// TwinCAT 3 PLC project PRG_Test_MachineControl
// ProgramVersion: 3.1.4024.0
// libraries:
//   B_Base, * (RafalOS)
//   B_IO, * (RafalOS)
//   B_MachineControl, * (RafalOS)
//   B_StatesAndModes, * (RafalOS)
//   Tc2_Standard, * (Beckhoff Automation GmbH)
//   Tc2_System, * (Beckhoff Automation GmbH)
//   Tc3_Module, * (Beckhoff Automation GmbH)
//   TcUnit, * (www.tcunit.org)
// project tree:
//   GVLs/ GVL_TestMCSafety.TcGVL, GVL_TestRequeestChange.TcGVL, GVL_TestSystemVariable.TcGVL, GVL_TopElement1.TcGVL, GVL_TopElement2.TcGVL, GVL_TestSaMContoller.TcGVL (not stored)
//   / PlcTask.TcTTO (not stored)
//   POUs/ FB_MyDefaultConfiguration.TcPOU, FB_MachineControl_NoneTE_Test.TcPOU, FB_MyNewConfigurationAddTE.TcPOU (not stored), FB_SaMControllerTest.TcPOU
//   POUs/POUs TopElement1/ FB_ControlElement1.TcPOU (not stored), FB_ControlElement2.TcPOU (not stored), FB_TopElement1.TcPOU, ITF_ControlElement1.TcIO (not stored), ITF_ControlElement2.TcIO (not stored), ITF_TopElement1.TcIO (not stored)
//   POUs/POUs TopElement2/ FB_ControlElement3.TcPOU (not stored), FB_ControlElement5.TcPOU, FB_ControlElement4.TcPOU (not stored), FB_ControlElement6.TcPOU, FB_GroupElement1.TcPOU, FB_TopElement2.TcPOU (not stored), ITF_ControlElement3.TcIO (not stored), ITF_ControlElement5.TcIO (not stored), ITF_ControlElement4.TcIO, ITF_ControlElement6.TcIO, ITF_GroupElement1.TcIO (not stored), ITF_TopElement2.TcIO (not stored)
//   TESTs/ PRG_Test.TcPOU (not stored)

// ---- GVLs/GVL_TestMCSafety.TcGVL
{attribute 'qualified_only'}
VAR_GLOBAL
	flSS1				: FB_BaseFlag;
	flSTO				: FB_BaseFlag;
	
END_VAR

// ---- GVLs/GVL_TestRequeestChange.TcGVL
{attribute 'qualified_only'}
VAR_GLOBAL
//Przyciski zmaiany stanu	
//	fbprUndefined			: FB_RequestChanges;
	fbprAbort				: FB_MCRequiredChange;
  	fbprClear				: FB_MCRequiredChange;
   	fbprReset				: FB_MCRequiredChange;
   	fbprStart				: FB_MCRequiredChange;
   	fbprStop				: FB_MCRequiredChange;
   	fbprHold				: FB_MCRequiredChange;
   	fbprUnhold				: FB_MCRequiredChange;
   	fbprSuspend				: FB_MCRequiredChange;
   	fbprUnsuspend			: FB_MCRequiredChange;
  	fbprComplete			: FB_MCRequiredChange;
//przyciski zmiany trybu
//	fbprNiedozwolony		: FB_SITP_PolecenieZmianyTrybu (ePolecenie := E_SITP_PolecenieZmianyTrybu.brak);     
	fbprProduction			: FB_MCRequiredChange;
    fbprMaintenance			: FB_MCRequiredChange;
    fbprManual				: FB_MCRequiredChange;
    fbprWashing				: FB_MCRequiredChange;
    fbprDiagnostics			: FB_MCRequiredChange;
//    fbprUzytkownika2		: FB_RequestChanges;
//   fbprUzytkownika3		: FB_RequestChanges;
//    fbprUzytkownika4		: FB_RequestChanges;
//    fbprUzytkownika5		: FB_RequestChanges;

END_VAR

// ---- GVLs/GVL_TestSystemVariable.TcGVL
{attribute 'qualified_only'}
VAR_GLOBAL
	fbTime							: FB_BaseTime;
	fbLocation						: FB_BaseLocation;
	fbLogger						: FB_BaseLogger;
	
	stCommonData					: ST_BaseCommonData;

	fbDefaultMachineConfiguration	: FB_MyDefaultConfiguration;
	fbMachineConfigure				: FB_MCMachineConfigure;
	
	fbSaMController					: FB_SaMController;
	
	fbMachineControl				: FB_MCMachineControl;
	
END_VAR

// ---- GVLs/GVL_TopElement1.TcGVL
{attribute 'qualified_only'}
VAR_GLOBAL
	senControlElement1Start		: FB_IOSensor_NO;
	senControlElement1End		: FB_IOSensor_NO;
	fbControlElement1			: FB_ControlElement1 (
									itfsenStart	:= senControlElement1Start,
	                                itfsenEnd	:= senControlElement1End
								);
	senControlElement2Start		: FB_IOSensor_NO;
	senControlElement2End		: FB_IOSensor_NO;
	senControlElement2Position1	: FB_IOSensor_NO;
	senControlElement2Position2	: FB_IOSensor_NO;
	fbControlElement2			:  FB_ControlElement2 (
									itfsenStart		:= senControlElement2Start,
	                                itfsenEnd		:= senControlElement2End,
	                                itfsenPosition1	:= senControlElement2Position1,
								    itfsenPosition2	:= senControlElement2Position2
								);

	senTopElement1Position1		: FB_IOSensor_NO;
	senTopElement1Position2		: FB_IOSensor_NO;
	fbTopElement1				: FB_TopElement1 (
									itfControlElement1		:= fbControlElement1,
								    itfControlElement2		:= fbControlElement2,
		                           	itfsenElementPosition1	:= senTopElement1Position1,
                                    itfsenElementPosition2	:= senTopElement1Position2
								);
END_VAR

// ---- GVLs/GVL_TopElement2.TcGVL
{attribute 'qualified_only'}
VAR_GLOBAL
	senControlElement3Start		: FB_IOSensor_NO;
	senControlElement3End		: FB_IOSensor_NO;
	fbControlElement3			: FB_ControlElement3 (
									itfsenStart	:= senControlElement3Start,
	                                itfsenEnd	:= senControlElement3End
								);
	senControlElement4Start		: FB_IOSensor_NO;
	senControlElement4End		: FB_IOSensor_NO;
	senControlElement4Position1	: FB_IOSensor_NO;
	senControlElement4Position2	: FB_IOSensor_NO;
	fbControlElement4			:  FB_ControlElement4 (
									itfsenStart		:= senControlElement4Start,
	                                itfsenEnd		:= senControlElement4End,
	                                itfsenPosition1	:= senControlElement4Position1,
								    itfsenPosition2	:= senControlElement4Position2
								);

	senGroupElement1Position1	: FB_IOSensor_NO;
	senGroupElement1Position2	: FB_IOSensor_NO;
	fbGroupElement1				: FB_GroupElement1 (
									itfControlElement3	:= fbControlElement3,
								    itfControlElement4	:= fbControlElement4,
								    itfsenPosition1		:= senGroupElement1Position1,
								    itfsenPosition2		:= senGroupElement1Position2
								);

	senControlElement5Start		: FB_IOSensor_NO;
	senControlElement5End		: FB_IOSensor_NO;
	fbControlElement5			: FB_ControlElement5 (
									itfsenStart	:= senControlElement5Start,
	                                itfsenEnd	:= senControlElement5End
								);
	senControlElement6Start		: FB_IOSensor_NO;
	senControlElement6End		: FB_IOSensor_NO;
	senControlElement6Position1	: FB_IOSensor_NO;
	senControlElement6Position2	: FB_IOSensor_NO;
	fbControlElement6			:  FB_ControlElement6 (
									itfsenStart		:= senControlElement6Start,
	                                itfsenEnd		:= senControlElement6End,
	                                itfsenPosition1	:= senControlElement6Position1,
								    itfsenPosition2	:= senControlElement6Position2
								);
								
								
	senTopElement1Position1		: FB_IOSensor_NO;
	senTopElement1Position2		: FB_IOSensor_NO;
	fbTopElement2				: FB_TopElement2 (
									itfGroupElement1		:= fbGroupElement1,
									itfControlElement5		:= fbControlElement5,
								    itfControlElement6		:= fbControlElement6,
		                           	itfsenElementPosition1	:= senTopElement1Position1,
                                    itfsenElementPosition2	:= senTopElement1Position2
								);
END_VAR

// ---- POUs/POUs TopElement2/ITF_ControlElement4.TcIO
INTERFACE ITF_ControlElement4 EXTENDS ITF_BaseControlElement

END_INTERFACE

// ---- POUs/POUs TopElement2/ITF_ControlElement6.TcIO
INTERFACE ITF_ControlElement6 EXTENDS ITF_BaseControlElement

END_INTERFACE

// ---- POUs/FB_MyDefaultConfiguration.TcPOU
FUNCTION_BLOCK FB_MyDefaultConfiguration EXTENDS FB_Base IMPLEMENTS ITF_MCConfiguration
VAR

END_VAR

METHOD PUBLIC AddTopElementToLogger : BOOL
VAR_INPUT
END_VAR
GVL_TestSystemVariable.fbMachineControl.JoinTheLogger ();
END_METHOD

(*			
	RafalOS
	Rafał Osajda		29.10.2025		TC 4024.66
	Dodawanie TopElementu do systemu
*)
METHOD PUBLIC AddTopElementToMachineControl : BOOL
VAR_INPUT
	itfMachineControl			: ITF_MCMachineControlConfigure;
END_VAR
THIS^.SetText (eLocation := E_BaseLocation.pl, wsDescription := "System");
THIS^.SetText (eLocation := E_BaseLocation.en, wsDescription := "System");
THIS^.SetText (eLocation := E_BaseLocation.de, wsDescription := "System");
GVL_TestSystemVariable.fbMachineControl.SetName (stName := THIS^.GetTexts ());
itfMachineControl.AddTopElementFromConfiguration (fbTopElement	:= GVL_TestSystemVariable.fbMachineControl);
END_METHOD

METHOD PUBLIC SetStartMode : BOOL
VAR_INPUT
	itfMachineControl			: ITF_MCMachineControlConfigure;
END_VAR
itfMachineControl.SetStartMode (eStartMode := E_BaseMachineMode.Production);
END_METHOD

METHOD StateAndModes : BOOL
VAR_INPUT
	itfMachineControl			: ITF_MCMachineControlConfigure;
END_VAR
itfMachineControl.AddRequestStateChange (iNumberOfRequest := E_SaMCommandChangeState.Clear,		itfRequest := GVL_TestRequeestChange.fbprClear);
itfMachineControl.AddRequestStateChange (iNumberOfRequest := E_SaMCommandChangeState.Reset, 	itfRequest := GVL_TestRequeestChange.fbprReset);
itfMachineControl.AddRequestStateChange (iNumberOfRequest := E_SaMCommandChangeState.Start, 	itfRequest := GVL_TestRequeestChange.fbprStart);
itfMachineControl.AddRequestStateChange (iNumberOfRequest := E_SaMCommandChangeState.Stop, 		itfRequest := GVL_TestRequeestChange.fbprStop);
itfMachineControl.AddRequestStateChange (iNumberOfRequest := E_SaMCommandChangeState.Suspend, 	itfRequest := GVL_TestRequeestChange.fbprSuspend);
itfMachineControl.AddRequestStateChange (iNumberOfRequest := E_SaMCommandChangeState.Unsuspend, itfRequest := GVL_TestRequeestChange.fbprUnsuspend);
itfMachineControl.AddRequestStateChange (iNumberOfRequest := E_SaMCommandChangeState.Hold, 		itfRequest := GVL_TestRequeestChange.fbprHold);
itfMachineControl.AddRequestStateChange (iNumberOfRequest := E_SaMCommandChangeState.Unhold, 	itfRequest := GVL_TestRequeestChange.fbprUnhold);
itfMachineControl.AddRequestStateChange (iNumberOfRequest := E_SaMCommandChangeState.Complete, 	itfRequest := GVL_TestRequeestChange.fbprComplete);
itfMachineControl.AddRequestStateChange (iNumberOfRequest := E_SaMCommandChangeState.Abort,		itfRequest := GVL_TestRequeestChange.fbprAbort);

itfMachineControl.AddRequestModeChange (iNumberOfRequest := E_SaMCommandChangeMode.Production, 	itfRequest := GVL_TestRequeestChange.fbprProduction);
itfMachineControl.AddRequestModeChange (iNumberOfRequest := E_SaMCommandChangeMode.Maintenance,	itfRequest := GVL_TestRequeestChange.fbprMaintenance);
itfMachineControl.AddRequestModeChange (iNumberOfRequest := E_SaMCommandChangeMode.Manual, 		itfRequest := GVL_TestRequeestChange.fbprManual);
itfMachineControl.AddRequestModeChange (iNumberOfRequest := E_SaMCommandChangeMode.Washing,		itfRequest := GVL_TestRequeestChange.fbprWashing);
itfMachineControl.AddRequestModeChange (iNumberOfRequest := E_SaMCommandChangeMode.Diagnostisc,	itfRequest := GVL_TestRequeestChange.fbprDiagnostics);
END_METHOD

END_FUNCTION_BLOCK

// ---- POUs/POUs TopElement1/FB_TopElement1.TcPOU
FUNCTION_BLOCK FB_TopElement1 EXTENDS FB_BaseTopElement IMPLEMENTS ITF_TopElement1
VAR
	itfControlElement1		: ITF_ControlElement1;
	itfControlElement2		: ITF_ControlElement2;
	itfsenElementPosition1	: ITF_IOSensor;
	itfsenElementPosition2	: ITF_IOSensor;
END_VAR

METHOD FB_init : BOOL
VAR_INPUT
	bInitRetains : BOOL; // if TRUE, the retain variables are initialized (warm start / cold start)
	bInCopyCode : BOOL;  // if TRUE, the instance afterwards gets moved into the copy code (online change)
	itfControlElement1		: ITF_ControlElement1;
	itfControlElement2		: ITF_ControlElement2;
	itfsenElementPosition1	: ITF_IOSensor;
	itfsenElementPosition2	: ITF_IOSensor;
END_VAR
THIS^.itfControlElement1			:= itfControlElement1;
THIS^.AddControlElement (itfControlElement	:= itfControlElement1);
THIS^.SetText (eLocation 			:= E_BaseLocation.pl, wsDescription := "Nazwa controlelementu 1 pl");
THIS^.SetText (eLocation 			:= E_BaseLocation.en, wsDescription := "Nazwa controlelementu 1 en");
THIS^.SetText (eLocation 			:= E_BaseLocation.de, wsDescription := "Nazwa controlelementu 1 de");
THIS^.itfControlElement1.SetName (stName	:= THIS^.GetTexts ());

THIS^.itfControlElement2			:= itfControlElement2;
THIS^.AddControlElement (itfControlElement	:= itfControlElement2);
THIS^.SetText (eLocation 			:= E_BaseLocation.pl, wsDescription := "Nazwa controlelementu 2 pl");
THIS^.SetText (eLocation 			:= E_BaseLocation.en, wsDescription := "Nazwa controlelementu 2 en");
THIS^.SetText (eLocation 			:= E_BaseLocation.de, wsDescription := "Nazwa controlelementu 2 de");
THIS^.itfControlElement2.SetName (stName	:= THIS^.GetTexts ());

THIS^.itfsenElementPosition1		:= itfsenElementPosition1;
THIS^.AddComponent (itfComponent	:= itfsenElementPosition1);
THIS^.SetText (eLocation 			:= E_BaseLocation.pl, wsDescription := "Nazwa komponentu 1 pl");
THIS^.SetText (eLocation 			:= E_BaseLocation.en, wsDescription := "Nazwa komponentu 1 en");
THIS^.SetText (eLocation 			:= E_BaseLocation.de, wsDescription := "Nazwa komponentu 1 de");
THIS^.itfsenElementPosition1.SetName (stName	:= THIS^.GetTexts ());

THIS^.itfsenElementPosition2		:= itfsenElementPosition2;
THIS^.AddComponent (itfComponent	:= itfsenElementPosition2);
THIS^.SetText (eLocation 			:= E_BaseLocation.pl, wsDescription := "Nazwa komponentu 2 pl");
THIS^.SetText (eLocation 			:= E_BaseLocation.en, wsDescription := "Nazwa komponentu 2 en");
THIS^.SetText (eLocation 			:= E_BaseLocation.de, wsDescription := "Nazwa komponentu 2 de");
THIS^.itfsenElementPosition2.SetName (stName	:= THIS^.GetTexts ());
END_METHOD

END_FUNCTION_BLOCK

// ---- POUs/POUs TopElement2/FB_GroupElement1.TcPOU
FUNCTION_BLOCK FB_GroupElement1 EXTENDS FB_BaseGroupElement IMPLEMENTS ITF_GroupElement1
VAR
	itfControlElement3		: ITF_ControlElement3;
	itfControlElement4		: ITF_ControlElement4;
	itfsenPosition1			: ITF_IOSensor;	
	itfsenPosition2			: ITF_IOSensor;	
END_VAR

METHOD FB_init : BOOL
VAR_INPUT
	bInitRetains : BOOL; // if TRUE, the retain variables are initialized (warm start / cold start)
	bInCopyCode : BOOL;  // if TRUE, the instance afterwards gets moved into the copy code (online change)
	itfControlElement3		: ITF_ControlElement3;
	itfControlElement4		: ITF_ControlElement4;
	itfsenPosition1			: ITF_IOSensor;	
	itfsenPosition2			: ITF_IOSensor;	
END_VAR
THIS^.itfControlElement3			:= itfControlElement3;
THIS^.AddControlElement (itfControlElement	:= itfControlElement3);
THIS^.SetText (eLocation 			:= E_BaseLocation.pl, wsDescription := "Nazwa control elementu 3 pl");
THIS^.SetText (eLocation 			:= E_BaseLocation.en, wsDescription := "Nazwa control elementu 3 en");
THIS^.SetText (eLocation 			:= E_BaseLocation.de, wsDescription := "Nazwa control elementu 3 de");
THIS^.itfControlElement3.SetName (stName	:= THIS^.GetTexts ());

THIS^.itfControlElement4			:= itfControlElement4;
THIS^.AddControlElement (itfControlElement	:= itfControlElement4);
THIS^.SetText (eLocation 			:= E_BaseLocation.pl, wsDescription := "Nazwa control elementu 4 2 pl");
THIS^.SetText (eLocation 			:= E_BaseLocation.en, wsDescription := "Nazwa control elementu 4 2 en");
THIS^.SetText (eLocation 			:= E_BaseLocation.de, wsDescription := "Nazwa control elementu 4 2 de");
THIS^.itfControlElement4.SetName (stName	:= THIS^.GetTexts ());

THIS^.itfsenPosition1				:= itfsenPosition1;
THIS^.AddComponent (itfComponent	:= itfsenPosition1);
THIS^.SetText (eLocation 			:= E_BaseLocation.pl, wsDescription := "Nazwa komponentu 3 pl");
THIS^.SetText (eLocation 			:= E_BaseLocation.en, wsDescription := "Nazwa komponentu 3 en");
THIS^.SetText (eLocation 			:= E_BaseLocation.de, wsDescription := "Nazwa komponentu 3 de");
THIS^.itfsenPosition1.SetName (stName	:= THIS^.GetTexts ());

THIS^.itfsenPosition2				:= itfsenPosition2;
THIS^.AddComponent (itfComponent	:= itfsenPosition2);
THIS^.SetText (eLocation 			:= E_BaseLocation.pl, wsDescription := "Nazwa komponentu 4 pl");
THIS^.SetText (eLocation 			:= E_BaseLocation.en, wsDescription := "Nazwa komponentu 4 en");
THIS^.SetText (eLocation 			:= E_BaseLocation.de, wsDescription := "Nazwa komponentu 4 de");
THIS^.itfsenPosition2.SetName (stName	:= THIS^.GetTexts ());
END_METHOD

END_FUNCTION_BLOCK

// ---- POUs/POUs TopElement2/FB_ControlElement5.TcPOU
FUNCTION_BLOCK FB_ControlElement5 EXTENDS FB_BaseControlElement IMPLEMENTS ITF_ControlElement5
VAR
	
	itfsenStart			: ITF_IOSensor;
	itfsenEnd			: ITF_IOSensor;	
END_VAR

METHOD FB_init : BOOL
VAR_INPUT
	bInitRetains : BOOL; // if TRUE, the retain variables are initialized (warm start / cold start)
	bInCopyCode : BOOL;  // if TRUE, the instance afterwards gets moved into the copy code (online change)
	itfsenStart			: ITF_IOSensor;
	itfsenEnd			: ITF_IOSensor;	
	
END_VAR
THIS^.itfsenStart					:= itfsenStart;
THIS^.AddComponent (itfComponent	:= itfsenStart);
THIS^.SetText (eLocation 			:= E_BaseLocation.pl, wsDescription := "Nazwa komponentu 1 pl");
THIS^.SetText (eLocation 			:= E_BaseLocation.en, wsDescription := "Nazwa komponentu 1 en");
THIS^.SetText (eLocation 			:= E_BaseLocation.de, wsDescription := "Nazwa komponentu 1 de");
THIS^.itfsenStart.SetName (stName	:= THIS^.GetTexts ());

THIS^.itfsenEnd						:= itfsenEnd;
THIS^.AddComponent (itfComponent	:= itfsenEnd);
THIS^.SetText (eLocation 			:= E_BaseLocation.pl, wsDescription := "Nazwa komponentu 2 pl");
THIS^.SetText (eLocation 			:= E_BaseLocation.en, wsDescription := "Nazwa komponentu 2 en");
THIS^.SetText (eLocation 			:= E_BaseLocation.de, wsDescription := "Nazwa komponentu 2 de");
THIS^.itfsenEnd.SetName (stName	:= THIS^.GetTexts ());
END_METHOD

END_FUNCTION_BLOCK

// ---- POUs/POUs TopElement2/FB_ControlElement6.TcPOU
FUNCTION_BLOCK FB_ControlElement6 EXTENDS FB_BaseControlElement IMPLEMENTS ITF_ControlElement6
VAR
	
	itfsenStart			: ITF_IOSensor;
	itfsenEnd			: ITF_IOSensor;	
	itfsenPosition1		: ITF_IOSensor;	
	itfsenPosition2		: ITF_IOSensor;	
END_VAR

METHOD FB_init : BOOL
VAR_INPUT
	bInitRetains : BOOL; // if TRUE, the retain variables are initialized (warm start / cold start)
	bInCopyCode : BOOL;  // if TRUE, the instance afterwards gets moved into the copy code (online change)
	itfsenStart			: ITF_IOSensor;
	itfsenEnd			: ITF_IOSensor;	
	itfsenPosition1		: ITF_IOSensor;	
	itfsenPosition2		: ITF_IOSensor;	
END_VAR
THIS^.itfsenStart					:= itfsenStart;
THIS^.AddComponent (itfComponent	:= itfsenStart);
THIS^.SetText (eLocation 			:= E_BaseLocation.pl, wsDescription := "Nazwa komponentu 1 pl");
THIS^.SetText (eLocation 			:= E_BaseLocation.en, wsDescription := "Nazwa komponentu 1 en");
THIS^.SetText (eLocation 			:= E_BaseLocation.de, wsDescription := "Nazwa komponentu 1 de");
THIS^.itfsenStart.SetName (stName	:= THIS^.GetTexts ());

THIS^.itfsenEnd						:= itfsenEnd;
THIS^.AddComponent (itfComponent	:= itfsenEnd);
THIS^.SetText (eLocation 			:= E_BaseLocation.pl, wsDescription := "Nazwa komponentu 2 pl");
THIS^.SetText (eLocation 			:= E_BaseLocation.en, wsDescription := "Nazwa komponentu 2 en");
THIS^.SetText (eLocation 			:= E_BaseLocation.de, wsDescription := "Nazwa komponentu 2 de");
THIS^.itfsenEnd.SetName (stName	:= THIS^.GetTexts ());

THIS^.itfsenPosition1				:= itfsenPosition1;
THIS^.AddComponent (itfComponent	:= itfsenPosition1);
THIS^.SetText (eLocation 			:= E_BaseLocation.pl, wsDescription := "Nazwa komponentu 3 pl");
THIS^.SetText (eLocation 			:= E_BaseLocation.en, wsDescription := "Nazwa komponentu 3 en");
THIS^.SetText (eLocation 			:= E_BaseLocation.de, wsDescription := "Nazwa komponentu 3 de");
THIS^.itfsenPosition1.SetName (stName	:= THIS^.GetTexts ());

THIS^.itfsenPosition2				:= itfsenPosition2;
THIS^.AddComponent (itfComponent	:= itfsenPosition2);
THIS^.SetText (eLocation 			:= E_BaseLocation.pl, wsDescription := "Nazwa komponentu 4 pl");
THIS^.SetText (eLocation 			:= E_BaseLocation.en, wsDescription := "Nazwa komponentu 4 en");
THIS^.SetText (eLocation 			:= E_BaseLocation.de, wsDescription := "Nazwa komponentu 4 de");
THIS^.itfsenPosition2.SetName (stName	:= THIS^.GetTexts ());
END_METHOD

END_FUNCTION_BLOCK

// ---- POUs/FB_MachineControl_NoneTE_Test.TcPOU
FUNCTION_BLOCK FB_MachineControl_NoneTE_Test EXTENDS TcUnit.FB_TestSuite
VAR
	bKoniec			: BOOL;
	iTest			: INT;
END_VAR

T01_FirstCycleInit ();
T02_FirstCycleMachine ();
//T03_PrzejsciePrzezStany ();


T99_Test ();

METHOD PRIVATE T01_FirstCycleInit
VAR_INPUT
END_VAR
IF (TcUnit.TEST_ORDERED ('T01_FirstCycleInit')) THEN
	iTest	:= 1;
	(*	Podpięcie zmiennych głównych do struktury	*)	
	GVL_TestSystemVariable.stCommonData.itfTime			:= GVL_TestSystemVariable.fbTime;
	GVL_TestSystemVariable.stCommonData.itfLocaciotn	:= GVL_TestSystemVariable.fbLocation;
	GVL_TestSystemVariable.stCommonData.itfLogger		:= GVL_TestSystemVariable.fbLogger;
	(*	Podpięcie zarządzania stanami i trybami pracy	*)
	GVL_TestSystemVariable.fbMachineControl.AddModulSaM (fbSaMController	:= GVL_TestSystemVariable.fbSaMController);
	(*	Podpięcie zmiennych Safety		*)
	GVL_TestSystemVariable.fbMachineControl.LinkSS1 (fbSS1	:= GVL_TestMCSafety.flSS1);
	GVL_TestSystemVariable.fbMachineControl.LinkSTO (fbSTO	:= GVL_TestMCSafety.flSTO);
	(*	Podpięcie podstawowej konfiguracji	*)
	GVL_TestSystemVariable.fbMachineControl.AddModulConfigure (fbMachineConfigure	:= GVL_TestSystemVariable.fbMachineConfigure);
	GVL_TestSystemVariable.fbMachineConfigure.AddConfiguration (fbConfigure := GVL_TestSystemVariable.fbDefaultMachineConfiguration);
	(*	Linkowanie zmiennych z modułami	*)
	GVL_TestSystemVariable.fbLogger.LinkCommonData (stCommonData 				:= GVL_TestSystemVariable.stCommonData);
	GVL_TestSystemVariable.fbMachineControl.LinkCommonData (stCommonData		:= GVL_TestSystemVariable.stCommonData);
	
	AssertEquals_INT (Expected := 1, Actual := GVL_TestSystemVariable.fbMachineConfigure.iNubmerOfAddedConfigure, Message := 'T01 - bledna ilosc konfiguracji');
	
	
	TcUnit.TEST_FINISHED ();
END_IF
END_METHOD

METHOD PRIVATE T02_FirstCycleMachine
VAR_INPUT
END_VAR
IF (TcUnit.TEST_ORDERED ('T02_FirstCycleMachine')) THEN
	iTest	:= 2;
	GVL_TestSystemVariable.fbMachineControl ();
	
	AssertEquals_UINT (Expected := 1, Actual := GVL_TestSystemVariable.fbMachineControl.uiNumberOfControlElement, Message := 'T01- bledna ilosc controlelementow');
	

	TcUnit.TEST_FINISHED ();
END_IF
END_METHOD

METHOD PRIVATE T20_PrzejsciePrzezStany
VAR_INST
	iStep			: INT;
	iStepChange		: INT;
	eModeExpected	: E_BaseMachineMode;
	eModeActual		: E_BaseMachineMode;
	eStateExpected	: E_BaseMachineState;
	eStateActual	: E_BaseMachineState;
END_VAR
IF (TcUnit.TEST_ORDERED ('T20_PrzejsciePrzezStany')) THEN
	GVL_TestSystemVariable.fbMachineControl ();
	CASE iStep OF
	0	:
		iTest := 3;
		GVL_TestSystemVariable.fbMachineControl ();
		GVL_TestMCSafety.flSS1.SetFlag (bState := TRUE);
        GVL_TestMCSafety.flSTO.SetFlag (bState := TRUE);
		WRITE_PROTECTED_INT (Ptr := ADR (GVL_TestSystemVariable.fbSaMController.eState), Value := 0);
		iStep := iStep + 10;
	10	:
		eModeActual := GVL_TestSystemVariable.fbSaMController.GetMode ();
		eModeExpected := E_BaseMachineMode.Production;
		AssertEquals (Expected := eModeExpected, Actual := eModeActual, Message := 'S10 - T01 - bledny tryb opuszczenie testu');
		IF (eModeExpected = eModeActual) THEN
			iStep		:= iStep + 10;
		ELSE
			iStep		:= GVL_BaseConstans.FINISH_STEP;
		END_IF
	20	:
		CASE iStepChange OF
		0	: eStateExpected := E_BaseMachineState.Aborting; 		GVL_TestRequeestChange.fbprAbort.SetRequiredChange (bIn := TRUE);
		1	: eStateExpected := E_BaseMachineState.Clearing;		GVL_TestRequeestChange.fbprClear.SetRequiredChange (bIN := TRUE);	//wyjscie z Aborted
		2	: eStateExpected := E_BaseMachineState.Resetting;		GVL_TestRequeestChange.fbprReset.SetRequiredChange (bIN := TRUE);
    	3	: eStateExpected := E_BaseMachineState.Starting;		GVL_TestRequeestChange.fbprStart.SetRequiredChange (bIN := TRUE);
		4	: eStateExpected := E_BaseMachineState.Suspending;		GVL_TestRequeestChange.fbprSuspend.SetRequiredChange (bIN := TRUE);
		5	: eStateExpected := E_BaseMachineState.Unsuspending;	GVL_TestRequeestChange.fbprUnsuspend.SetRequiredChange (bIN := TRUE);
		6	: eStateExpected := E_BaseMachineState.Holding;			GVL_TestRequeestChange.fbprHold.SetRequiredChange (bIN := TRUE);
		7	: eStateExpected := E_BaseMachineState.Unholding;		GVL_TestRequeestChange.fbprUnhold.SetRequiredChange (bIN := TRUE);
		8	: eStateExpected := E_BaseMachineState.Completing;		GVL_TestRequeestChange.fbprComplete.SetRequiredChange (bIN := TRUE);
		9	: eStateExpected := E_BaseMachineState.Resetting;		GVL_TestRequeestChange.fbprReset.SetRequiredChange (bIN := TRUE);
		10	: eStateExpected := E_BaseMachineState.Stopping;		GVL_TestRequeestChange.fbprStop.SetRequiredChange (bIN := TRUE);
		11	: eStateExpected := E_BaseMachineState.Aborting;		GVL_TestRequeestChange.fbprAbort.SetRequiredChange (bIN := TRUE);	//petla zrobiona dojcie jeszcze raz to execute
		12	: eStateExpected := E_BaseMachineState.Clearing;		GVL_TestRequeestChange.fbprClear.SetRequiredChange (bIN := TRUE);
		13	: eStateExpected := E_BaseMachineState.Resetting;		GVL_TestRequeestChange.fbprReset.SetRequiredChange (bIN := TRUE);
    	14	: eStateExpected := E_BaseMachineState.Starting;		GVL_TestRequeestChange.fbprStart.SetRequiredChange (bIN := TRUE);
		15	: eStateExpected := E_BaseMachineState.Stopping;		GVL_TestRequeestChange.fbprStop.SetRequiredChange (bIN := TRUE);	//i nacisniecie stop
		16	: eStateExpected := E_BaseMachineState.Resetting;		GVL_TestRequeestChange.fbprReset.SetRequiredChange (bIN := TRUE);	//Dojscie jeszcze raz do execute
    	17	: eStateExpected := E_BaseMachineState.Starting;		GVL_TestRequeestChange.fbprStart.SetRequiredChange (bIN := TRUE);
		18	: eStateExpected := E_BaseMachineState.Aborting;		GVL_TestRequeestChange.fbprAbort.SetRequiredChange (bIN := TRUE);	//i nacisniecie grzyba
		END_CASE
		iStepChange := iStepChange + 1;	
		iStep := iStep + 10;
	30	:
		AssertTrue (Condition := 	GVL_TestSystemVariable.fbSaMController.IsChangeStateBusy (), 	Message := 'S30 - T01 - Bledny stan busy');
		AssertFalse (Condition := 	GVL_TestSystemVariable.fbSaMController.IsChangeStateDone (), 	Message := 'S30 - T02 - Bledny stan done');
		AssertFalse (Condition := 	GVL_TestSystemVariable.fbSaMController.IsChangeStateStatus (), 	Message := 'S30 - T03 - Bledny stan status');
		iStep	:= iStep + 10;
	40	://krok zmiany stanu
		AssertTrue (Condition := 	GVL_TestSystemVariable.fbSaMController.IsChangeStateBusy (), 	Message := 'S40 - T01 - Bledny stan busy');
		AssertFalse (Condition := 	GVL_TestSystemVariable.fbSaMController.IsChangeStateDone (),	Message := 'S40 - T02 - Bledny stan done');
		AssertFalse (Condition := 	GVL_TestSystemVariable.fbSaMController.IsChangeStateStatus (), 	Message := 'S40 - T03 - Bledny stan status');
		iStep	:= iStep + 10;
	50	:	//ostani krok 
		AssertFalse (Condition := 	GVL_TestSystemVariable.fbSaMController.IsChangeStateBusy (), 	Message := 'S50 - T01 - Bledny stan busy');
		AssertTrue (Condition := 	GVL_TestSystemVariable.fbSaMController.IsChangeStateDone (), 	Message := 'S50 - T02 - Bledny stan done');
		AssertTrue (Condition := 	GVL_TestSystemVariable.fbSaMController.IsChangeStateStatus (), 	Message := 'S50 - T03 - Bledny stan status');
		iStep	:= iStep + 10;
	60	:
		eStateActual			:= GVL_TestSystemVariable.fbSaMController.GetState ();
		AssertEquals_INT (Expected := eStateExpected, Actual := eStateActual, Message := 'S60 - T01 - Bledny stan');
		IF (eStateExpected <> eStateActual) THEN
			AssertFalse (Condition := TRUE, Message := 'S60 - T02 - Wyjscie przy blednym stanie');
			iStep				:= GVL_BaseConstans.FINISH_STEP;
		ELSE
			CASE eStateActual OF
				E_BaseMachineState.Aborting		: eStateExpected	:= E_BaseMachineState.Aborted;
				E_BaseMachineState.Clearing		: eStateExpected	:= E_BaseMachineState.Stopped;
				E_BaseMachineState.Stopping		: eStateExpected	:= E_BaseMachineState.Stopped;
				E_BaseMachineState.Resetting	: eStateExpected	:= E_BaseMachineState.Idle;
				E_BaseMachineState.Starting		: eStateExpected	:= E_BaseMachineState.Execute;
				E_BaseMachineState.Unsuspending	: eStateExpected	:= E_BaseMachineState.Execute;
				E_BaseMachineState.Unholding	: eStateExpected	:= E_BaseMachineState.Execute;
				E_BaseMachineState.Suspending	: eStateExpected	:= E_BaseMachineState.Suspended;
				E_BaseMachineState.Holding		: eStateExpected	:= E_BaseMachineState.Held;
				E_BaseMachineState.Completing	: eStateExpected	:= E_BaseMachineState.Complete;
			END_CASE
//			iStep				:= iStep + 10;
//		END_IF
//	70	:
			AssertTrue (Condition := 	GVL_TestSystemVariable.fbSaMController.IsChangeStateBusy (), 	Message := 'S60 - T01 - Bledny stan busy');
			AssertFalse (Condition := 	GVL_TestSystemVariable.fbSaMController.IsChangeStateDone (), 	Message := 'S60 - T02 - Bledny stan done');
			AssertFalse (Condition := 	GVL_TestSystemVariable.fbSaMController.IsChangeStateStatus (), 	Message := 'S60 - T03 - Bledny stan status');
			iStep	:= iStep + 10;
		END_IF
	70	://krok zmiany stanu
		AssertTrue (Condition := 	GVL_TestSystemVariable.fbSaMController.IsChangeStateBusy (), 	Message := 'S70 - T01 - Bledny stan busy');
		AssertFalse (Condition := 	GVL_TestSystemVariable.fbSaMController.IsChangeStateDone (),	Message := 'S70 - T02 - Bledny stan done');
		AssertFalse (Condition := 	GVL_TestSystemVariable.fbSaMController.IsChangeStateStatus (), 	Message := 'S70 - T03 - Bledny stan status');
		iStep	:= iStep + 10;
	80	:	//ostani krok 
		AssertFalse (Condition := 	GVL_TestSystemVariable.fbSaMController.IsChangeStateBusy (), 	Message := 'S80 - T01 - Bledny stan busy');
		AssertTrue (Condition := 	GVL_TestSystemVariable.fbSaMController.IsChangeStateDone (), 	Message := 'S80 - T02 - Bledny stan done');
		AssertTrue (Condition :=	GVL_TestSystemVariable.fbSaMController.IsChangeStateStatus (), 	Message := 'S80 - T03 - Bledny stan status');
		iStep	:= iStep + 10;
	90	:
		eStateActual			:= GVL_TestSystemVariable.fbSaMController.GetState ();
		AssertEquals_INT (Expected := eStateExpected, Actual := eStateActual, Message := 'S100 - T01 - Bledny stan');
		IF (eStateExpected <> eStateActual) THEN
			AssertFalse (Condition := TRUE, Message := 'S100 - T02 - Wyjscie przy blednym stanie');
			iStep				:= GVL_BaseConstans.FINISH_STEP;
		ELSE
			IF (iStepChange = 19) THEN
				iStep				:= GVL_BaseConstans.FINISH_STEP;
			ELSE
				iStep				:= 20;
			END_IF
		END_IF	
	GVL_BaseConstans.FINISH_STEP	:
		TcUnit.TEST_FINISHED ();
	END_CASE
END_IF
END_METHOD

METHOD PRIVATE T99_Test
VAR_INPUT
END_VAR
IF (TcUnit.TEST_ORDERED ('T99_Test')) THEN
	IF (iTest <> 99) THEN
		iTest	:= 99;
		GVL_TestMCSafety.flSS1.SetFlag (bState := TRUE);
		GVL_TestMCSafety.flSTO.SetFlag (bState := TRUE);
	END_IF
	GVL_TestSystemVariable.fbMachineControl ();
	IF (bKoniec) THEN
		bKoniec	:= FALSE;
		TcUnit.TEST_FINISHED ();
	END_IF
END_IF
END_METHOD

END_FUNCTION_BLOCK

// ---- POUs/FB_SaMControllerTest.TcPOU
FUNCTION_BLOCK FB_SaMControllerTest EXTENDS TcUnit.FB_TestSuite
VAR
	iTest			: INT;
END_VAR

T01_WiazanieZmiennych ();
T02_PrzelaczanieTrybow ();
T03_PrzelaczanieStanow ();

METHOD PROTECTED T01_WiazanieZmiennych
VAR_INPUT
END_VAR
IF (TcUnit.TEST_ORDERED ('T01_WiazanieZmiennych')) THEN
	itest	:= 1;
	
	GVL_TestSaMContoller.stCommonData.itfTime			:= GVL_TestSaMContoller.fbTime;
	GVL_TestSaMContoller.stCommonData.itfLocaciotn		:= GVL_TestSaMContoller.fbLocation;
	GVL_TestSaMContoller.stCommonData.itfLogger			:= GVL_TestSaMContoller.fbLogger;

	GVL_TestSaMContoller.fbMySaMController.LinkSS1 (fbSS1	:= GVL_TestSaMContoller.flSS1);
	GVL_TestSaMContoller.fbMySaMController.LinkSTO (fbSTO	:= GVL_TestSaMContoller.flSTO);

	GVL_TestSaMContoller.fbMySaMController.LinkCommonData (stCommonData	:= GVL_TestSaMContoller.stCommonData);

	AssertEquals_UINT (Expected := 129, Actual := GVL_TestSaMContoller.fbMySaMController.uiNumberOfComponents, Message := 'T01 - bledna libcza lkomponentow');
	
	
	TcUnit.TEST_FINISHED ();
END_IF
END_METHOD

METHOD PRIVATE T02_PrzelaczanieTrybow
VAR_INST
	iStep			: INT;
	eNewMode		: E_BaseMachineMode;
	eActualMode		: E_BaseMachineMode;
	
END_VAR
IF (TcUnit.TEST_ORDERED ('T02_PrzelaczanieTrybow')) THEN
	GVL_TestSaMContoller.fbMySaMController.ExecuteEveryCycle_Test ();
	GVL_TestSaMContoller.fbMySaMController.ExecuteEveryCycle_Operation ();
	GVL_TestSaMContoller.fbMySaMController.ExecuteEveryCycle_Status ();
	GVL_TestSaMContoller.fbMySaMController.ExecuteEveryCycle_Error ();
	CASE iStep OF
	0	:
		itest	:= 3;
		eNewMode			:= E_BaseMachineMode.Production;
		GVL_TestSaMContoller.fbMySaMController.Execute (iNumberOfCommand := eNewMode, eChangeCategory := E_SaMChangeCategory.eMode);
		iStep	:= iStep + 10;
	10	:	//pierwszy krok 
		AssertTrue (Condition := GVL_TestSaMContoller.fbMySaMController.IsChangeModeBusy (), 	Message := 'S10 - T01 - Bledny stan busy');
		AssertFalse (Condition := GVL_TestSaMContoller.fbMySaMController.IsChangeModeDone (), 	Message := 'S10 - T02 - Bledny stan done');
		AssertFalse (Condition := GVL_TestSaMContoller.fbMySaMController.IsChangeModeStatus (), Message := 'S10 - T03 - Bledny stan status');
		iStep	:= iStep + 10;
	20	://krok zmiany stanu
		AssertTrue (Condition := GVL_TestSaMContoller.fbMySaMController.IsChangeModeBusy (), 	Message := 'S20 - T01 - Bledny stan busy');
		AssertFalse (Condition := GVL_TestSaMContoller.fbMySaMController.IsChangeModeDone (),	Message := 'S20 - T02 - Bledny stan done');
		AssertFalse (Condition := GVL_TestSaMContoller.fbMySaMController.IsChangeModeStatus (), Message := 'S20 - T03 - Bledny stan status');
		iStep	:= iStep + 10;
	30	:	//ostani krok 
		AssertFalse (Condition := GVL_TestSaMContoller.fbMySaMController.IsChangeModeBusy (), 	Message := 'S30 - T01 - Bledny stan busy');
		AssertTrue (Condition := GVL_TestSaMContoller.fbMySaMController.IsChangeModeDone (), 	Message := 'S30 - T02 - Bledny stan done');
		AssertTrue (Condition := GVL_TestSaMContoller.fbMySaMController.IsChangeModeStatus (), 	Message := 'S30 - T03 - Bledny stan status');
		eActualMode				:= GVL_TestSaMContoller.fbMySaMController.GetMode ();
		AssertEquals (Expected := eNewMode, Actual := eActualMode, 						Message := 'S30 - T04 - Bledny stan');
		iStep	:= iStep + 10;
	40	:
		iStep	:= iStep + 10;
	50	:
		eNewMode			:= E_BaseMachineMode.Maintenance;
		GVL_TestSaMContoller.fbMySaMController.Execute (iNumberOfCommand := eNewMode, eChangeCategory := E_SaMChangeCategory.eMode);
		iStep	:= iStep + 10;
	60	:	//pierwszy krok 
		AssertTrue (Condition := GVL_TestSaMContoller.fbMySaMController.IsChangeModeBusy (), 	Message := 'S60 - T01 - Bledny stan busy');
		AssertFalse (Condition := GVL_TestSaMContoller.fbMySaMController.IsChangeModeDone (), 	Message := 'S60 - T02 - Bledny stan done');
		AssertFalse (Condition := GVL_TestSaMContoller.fbMySaMController.IsChangeModeStatus (), Message := 'S60 - T03 - Bledny stan status');
		iStep	:= iStep + 10;
	70	://krok zmiany stanu
		AssertTrue (Condition := GVL_TestSaMContoller.fbMySaMController.IsChangeModeBusy (), 	Message := 'S70 - T01 - Bledny stan busy');
		AssertFalse (Condition := GVL_TestSaMContoller.fbMySaMController.IsChangeModeDone (),	Message := 'S70 - T02 - Bledny stan done');
		AssertFalse (Condition := GVL_TestSaMContoller.fbMySaMController.IsChangeModeStatus (), Message := 'S70 - T03 - Bledny stan status');
		iStep	:= iStep + 10;
	80	:	//ostani krok 
		AssertFalse (Condition := GVL_TestSaMContoller.fbMySaMController.IsChangeModeBusy (), 	Message := 'S80 - T01 - Bledny stan busy');
		AssertTrue (Condition := GVL_TestSaMContoller.fbMySaMController.IsChangeModeDone (), 	Message := 'S80 - T02 - Bledny stan done');
		AssertTrue (Condition := GVL_TestSaMContoller.fbMySaMController.IsChangeModeStatus (), 	Message := 'S80 - T03 - Bledny stan status');
		eActualMode				:= GVL_TestSaMContoller.fbMySaMController.GetMode ();
		AssertEquals (Expected := eNewMode, Actual := eActualMode, 						Message := 'S80 - T04 - Bledny stan');
		iStep	:= iStep + 10;
	90	:
		iStep	:= iStep + 10;
	100	:
		eNewMode			:= E_BaseMachineMode.Manual;
		GVL_TestSaMContoller.fbMySaMController.Execute (iNumberOfCommand := eNewMode, eChangeCategory := E_SaMChangeCategory.eMode);
		iStep	:= iStep + 10;
	110	:	//pierwszy krok 
		AssertTrue (Condition := GVL_TestSaMContoller.fbMySaMController.IsChangeModeBusy (), 	Message := 'S110 - T01 - Bledny stan busy');
		AssertFalse (Condition := GVL_TestSaMContoller.fbMySaMController.IsChangeModeDone (), 	Message := 'S110 - T02 - Bledny stan done');
		AssertFalse (Condition := GVL_TestSaMContoller.fbMySaMController.IsChangeModeStatus (), Message := 'S110 - T03 - Bledny stan status');
		iStep	:= iStep + 10;
	120	://krok zmiany stanu
		AssertTrue (Condition := GVL_TestSaMContoller.fbMySaMController.IsChangeModeBusy (), 	Message := 'S120 - T01 - Bledny stan busy');
		AssertFalse (Condition := GVL_TestSaMContoller.fbMySaMController.IsChangeModeDone (),	Message := 'S120 - T02 - Bledny stan done');
		AssertFalse (Condition := GVL_TestSaMContoller.fbMySaMController.IsChangeModeStatus (), Message := 'S120 - T03 - Bledny stan status');
		iStep	:= iStep + 10;
	130	:	//ostani krok 
		AssertFalse (Condition := GVL_TestSaMContoller.fbMySaMController.IsChangeModeBusy (), 	Message := 'S130 - T01 - Bledny stan busy');
		AssertTrue (Condition := GVL_TestSaMContoller.fbMySaMController.IsChangeModeDone (), 	Message := 'S130 - T02 - Bledny stan done');
		AssertTrue (Condition := GVL_TestSaMContoller.fbMySaMController.IsChangeModeStatus (), 	Message := 'S130 - T03 - Bledny stan status');
		eActualMode				:= GVL_TestSaMContoller.fbMySaMController.GetMode ();
		AssertEquals (Expected := eNewMode, Actual := eActualMode, 						Message := 'S130 - T04 - Bledny stan');
		iStep	:= iStep + 10;
	140	:
		iStep	:= iStep + 10;
	150	:
		eNewMode			:= E_BaseMachineMode.Production;
		GVL_TestSaMContoller.fbMySaMController.Execute (iNumberOfCommand := eNewMode, eChangeCategory := E_SaMChangeCategory.eMode);
		iStep	:= iStep + 10;
	160	:	//pierwszy krok 
		AssertTrue (Condition := GVL_TestSaMContoller.fbMySaMController.IsChangeModeBusy (), 	Message := 'S160 - T01 - Bledny stan busy');
		AssertFalse (Condition := GVL_TestSaMContoller.fbMySaMController.IsChangeModeDone (), 	Message := 'S160 - T02 - Bledny stan done');
		AssertFalse (Condition := GVL_TestSaMContoller.fbMySaMController.IsChangeModeStatus (), Message := 'S160 - T03 - Bledny stan status');
		iStep	:= iStep + 10;
	170	://krok zmiany stanu
		AssertTrue (Condition := GVL_TestSaMContoller.fbMySaMController.IsChangeModeBusy (), 	Message := 'S170 - T01 - Bledny stan busy');
		AssertFalse (Condition := GVL_TestSaMContoller.fbMySaMController.IsChangeModeDone (),	Message := 'S170 - T02 - Bledny stan done');
		AssertFalse (Condition := GVL_TestSaMContoller.fbMySaMController.IsChangeModeStatus (), Message := 'S170 - T03 - Bledny stan status');
		iStep	:= iStep + 10;
	180	:	//ostani krok 
		AssertFalse (Condition := GVL_TestSaMContoller.fbMySaMController.IsChangeModeBusy (), 	Message := 'S180 - T01 - Bledny stan busy');
		AssertTrue (Condition := GVL_TestSaMContoller.fbMySaMController.IsChangeModeDone (), 	Message := 'S180 - T02 - Bledny stan done');
		AssertTrue (Condition := GVL_TestSaMContoller.fbMySaMController.IsChangeModeStatus (), 	Message := 'S180 - T03 - Bledny stan status');
		eActualMode				:= GVL_TestSaMContoller.fbMySaMController.GetMode ();
		AssertEquals (Expected := eNewMode, Actual := eActualMode, 						Message := 'S180 - T04 - Bledny stan');
		iStep	:= iStep + 10;
	190	:	//jest w produkcji wyłączamy manual i próba wejścia 
		GVL_TestSaMContoller.fbMySaMController.SetModeEnabled (iMode := E_BaseMachineMode.Manual, bValue := FALSE);
		iStep	:= iStep + 10;
	200	:
		eNewMode			:= E_BaseMachineMode.Manual;
		GVL_TestSaMContoller.fbMySaMController.Execute (iNumberOfCommand := eNewMode, eChangeCategory := E_SaMChangeCategory.eMode);
		iStep	:= iStep + 10;
	210	:	//pierwszy krok 
		Assertfalse (Condition := GVL_TestSaMContoller.fbMySaMController.IsChangeModeBusy (), 	Message := 'S210 - T01 - Bledny stan busy');
		AssertTrue (Condition := GVL_TestSaMContoller.fbMySaMController.IsChangeModeDone (), 	Message := 'S210 - T02 - Bledny stan done');
		AssertTrue (Condition := GVL_TestSaMContoller.fbMySaMController.IsChangeModeStatus (), Message := 'S210 - T03 - Bledny stan status');
		iStep	:= iStep + 10;
	220	:	//jest w produkcji włączamy manual i próba wejścia 
		GVL_TestSaMContoller.fbMySaMController.SetModeEnabled (iMode := E_BaseMachineMode.Manual, bValue := TRUE);
		iStep	:= iStep + 10;
	230	:
		eNewMode			:= E_BaseMachineMode.Manual;
		GVL_TestSaMContoller.fbMySaMController.Execute (iNumberOfCommand := eNewMode, eChangeCategory := E_SaMChangeCategory.eMode);
		iStep	:= iStep + 10;
	240	:	//pierwszy krok 
		AssertTrue (Condition := GVL_TestSaMContoller.fbMySaMController.IsChangeModeBusy (), 	Message := 'S240 - T01 - Bledny stan busy');
		AssertFalse (Condition := GVL_TestSaMContoller.fbMySaMController.IsChangeModeDone (), 	Message := 'S240 - T02 - Bledny stan done');
		AssertFalse (Condition := GVL_TestSaMContoller.fbMySaMController.IsChangeModeStatus (), Message := 'S240 - T03 - Bledny stan status');
		iStep	:= iStep + 10;
	250	://krok zmiany stanu
		AssertTrue (Condition := GVL_TestSaMContoller.fbMySaMController.IsChangeModeBusy (), 	Message := 'S250 - T01 - Bledny stan busy');
		AssertFalse (Condition := GVL_TestSaMContoller.fbMySaMController.IsChangeModeDone (),	Message := 'S250 - T02 - Bledny stan done');
		AssertFalse (Condition := GVL_TestSaMContoller.fbMySaMController.IsChangeModeStatus (), Message := 'S250 - T03 - Bledny stan status');
		iStep	:= iStep + 10;
	260	:	//ostani krok 
		AssertFalse (Condition := GVL_TestSaMContoller.fbMySaMController.IsChangeModeBusy (), 	Message := 'S260 - T01 - Bledny stan busy');
		AssertTrue (Condition := GVL_TestSaMContoller.fbMySaMController.IsChangeModeDone (), 	Message := 'S260 - T02 - Bledny stan done');
		AssertTrue (Condition := GVL_TestSaMContoller.fbMySaMController.IsChangeModeStatus (), 	Message := 'S260 - T03 - Bledny stan status');
		eActualMode				:= GVL_TestSaMContoller.fbMySaMController.GetMode ();
		AssertEquals (Expected := eNewMode, Actual := eActualMode, 						Message := 'S260 - T04 - Bledny stan');
		iStep	:= iStep + 10;
	270	:
		eNewMode			:= E_BaseMachineMode.Production;
		GVL_TestSaMContoller.fbMySaMController.Execute (iNumberOfCommand := eNewMode, eChangeCategory := E_SaMChangeCategory.eMode);
		iStep	:= iStep + 10;
	280	:	//pierwszy krok 
		iStep	:= iStep + 10;
	290	://krok zmiany stanu
		iStep	:= iStep + 10;
	300	:	//ostani krok 
		eActualMode				:= GVL_TestSaMContoller.fbMySaMController.GetMode ();
		AssertEquals (Expected := eNewMode, Actual := eActualMode, 						Message := 'S300 - T04 - Bledny stan');
		iStep	:= iStep + 10;
	310	:
		TcUnit.TEST_FINISHED ();
	END_CASE	
END_IF
END_METHOD

METHOD PRIVATE T03_PrzelaczanieStanow
VAR_INST
	iStep			: INT;
	eNewState		: E_BaseMachineState;
	eActualState	: E_BaseMachineState;

END_VAR
IF (TcUnit.TEST_ORDERED ('T04_TestZmianyStanow')) THEN
	GVL_TestSaMContoller.fbMySaMController.ExecuteEveryCycle_Test ();
	GVL_TestSaMContoller.fbMySaMController.ExecuteEveryCycle_Operation ();
	GVL_TestSaMContoller.fbMySaMController.ExecuteEveryCycle_Status ();
	GVL_TestSaMContoller.fbMySaMController.ExecuteEveryCycle_Error ();
	CASE iStep OF
	0	:
		itest	:= 4;
(*	*)	eNewState			:= E_BaseMachineState.Aborting;
		GVL_TestSaMContoller.fbMySaMController.Execute (iNumberOfCommand := E_SaMCommandChangeState.Abort, eChangeCategory := E_SaMChangeCategory.eState);
		iStep	:= iStep + 10;
	10	:	//pierwszy krok 
		AssertTrue (Condition := GVL_TestSaMContoller.fbMySaMController.IsChangeStateBusy (), 		Message := 'S10 - T01 - Bledny stan busy');
		AssertFalse (Condition := GVL_TestSaMContoller.fbMySaMController.IsChangeStateDone (), 		Message := 'S10 - T02 - Bledny stan done');
		AssertFalse (Condition := GVL_TestSaMContoller.fbMySaMController.IsChangeStateStatus (), 	Message := 'S10 - T03 - Bledny stan status');
		iStep	:= iStep + 10;
	20	://krok zmiany stanu
		AssertTrue (Condition := GVL_TestSaMContoller.fbMySaMController.IsChangeStateBusy (), 		Message := 'S20 - T01 - Bledny stan busy');
		AssertFalse (Condition := GVL_TestSaMContoller.fbMySaMController.IsChangeStateDone (),		Message := 'S20 - T02 - Bledny stan done');
		AssertFalse (Condition := GVL_TestSaMContoller.fbMySaMController.IsChangeStateStatus (), 	Message := 'S20 - T03 - Bledny stan status');
		iStep	:= iStep + 10;
	30	:	//ostani krok 
		AssertFalse (Condition := GVL_TestSaMContoller.fbMySaMController.IsChangeStateBusy (), 		Message := 'S30 - T01 - Bledny stan busy');
		AssertTrue (Condition := GVL_TestSaMContoller.fbMySaMController.IsChangeStateDone (), 		Message := 'S30 - T02 - Bledny stan done');
		AssertTrue (Condition := GVL_TestSaMContoller.fbMySaMController.IsChangeStateStatus (), 	Message := 'S30 - T03 - Bledny stan status');
		eActualState				:= GVL_TestSaMContoller.fbMySaMController.GetState ();
		AssertEquals (Expected := eNewState, Actual := eActualState, 						Message := 'S30 - T04 - Bledny stan');
		iStep	:= iStep + 10;
	40	:
		iStep	:= iStep + 10;
	50	:	
(*	*)	eNewState	:= E_BaseMachineState.Aborted;
		GVL_TestSaMContoller.fbMySaMController.ChangeStateTo (eNewState := eNewState);
		iStep	:= iStep + 10;
	60	:	//pierwszy krok 
		AssertTrue (Condition := GVL_TestSaMContoller.fbMySaMController.IsChangeStateBusy (), 		Message := 'S60 - T01 - Bledny stan busy');
		AssertFalse (Condition := GVL_TestSaMContoller.fbMySaMController.IsChangeStateDone (), 		Message := 'S60 - T02 - Bledny stan done');
		AssertFalse (Condition := GVL_TestSaMContoller.fbMySaMController.IsChangeStateStatus (), 	Message := 'S60 - T03 - Bledny stan status');
		iStep	:= iStep + 10;
	70	://krok zmiany stanu
		AssertTrue (Condition := GVL_TestSaMContoller.fbMySaMController.IsChangeStateBusy (), 		Message := 'S70 - T01 - Bledny stan busy');
		AssertFalse (Condition := GVL_TestSaMContoller.fbMySaMController.IsChangeStateDone (),		Message := 'S70 - T02 - Bledny stan done');
		AssertFalse (Condition := GVL_TestSaMContoller.fbMySaMController.IsChangeStateStatus (), 	Message := 'S70 - T03 - Bledny stan status');
		iStep	:= iStep + 10;
	80	:	//ostani krok 
		AssertFalse (Condition := GVL_TestSaMContoller.fbMySaMController.IsChangeStateBusy (), 		Message := 'S80 - T01 - Bledny stan busy');
		AssertTrue (Condition := GVL_TestSaMContoller.fbMySaMController.IsChangeStateDone (), 		Message := 'S80 - T02 - Bledny stan done');
		AssertTrue (Condition := GVL_TestSaMContoller.fbMySaMController.IsChangeStateStatus (), 	Message := 'S80 - T03 - Bledny stan status');
		eActualState				:= GVL_TestSaMContoller.fbMySaMController.GetState ();
		AssertEquals (Expected := eNewState, Actual := eActualState, 						Message := 'S80 - T04 - Bledny stan');
		iStep	:= iStep + 10;
	90	:
		iStep	:= iStep + 10;
	100	:
(*	*)	eNewState			:= E_BaseMachineState.Clearing;
		GVL_TestSaMContoller.fbMySaMController.Execute (iNumberOfCommand := E_SaMCommandChangeState.Clear, eChangeCategory := E_SaMChangeCategory.eState);
		iStep	:= iStep + 10;
	110	:	//pierwszy krok 
		AssertTrue (Condition := GVL_TestSaMContoller.fbMySaMController.IsChangeStateBusy (), 		Message := 'S110 - T01 - Bledny stan busy');
		AssertFalse (Condition := GVL_TestSaMContoller.fbMySaMController.IsChangeStateDone (), 		Message := 'S110 - T02 - Bledny stan done');
		AssertFalse (Condition := GVL_TestSaMContoller.fbMySaMController.IsChangeStateStatus (), 	Message := 'S110 - T03 - Bledny stan status');
		iStep	:= iStep + 10;
	120	://krok zmiany stanu
		AssertTrue (Condition := GVL_TestSaMContoller.fbMySaMController.IsChangeStateBusy (), 		Message := 'S120 - T01 - Bledny stan busy');
		AssertFalse (Condition := GVL_TestSaMContoller.fbMySaMController.IsChangeStateDone (),		Message := 'S120 - T02 - Bledny stan done');
		AssertFalse (Condition := GVL_TestSaMContoller.fbMySaMController.IsChangeStateStatus (), 	Message := 'S120 - T03 - Bledny stan status');
		iStep	:= iStep + 10;
	130	:	//ostani krok 
		AssertFalse (Condition := GVL_TestSaMContoller.fbMySaMController.IsChangeStateBusy (), 		Message := 'S130 - T01 - Bledny stan busy');
		AssertTrue (Condition := GVL_TestSaMContoller.fbMySaMController.IsChangeStateDone (), 		Message := 'S130 - T02 - Bledny stan done');
		AssertTrue (Condition := GVL_TestSaMContoller.fbMySaMController.IsChangeStateStatus (), 	Message := 'S130 - T03 - Bledny stan status');
		eActualState				:= GVL_TestSaMContoller.fbMySaMController.GetState ();
		AssertEquals (Expected := eNewState, Actual := eActualState, 						Message := 'S130 - T04 - Bledny stan');
		iStep	:= iStep + 10;
	140	:
		iStep	:= iStep + 10;
	150	:
(*	*)	eNewState			:= E_BaseMachineState.Stopped;
		GVL_TestSaMContoller.fbMySaMController.ChangeStateTo (eNewState := eNewState);
		iStep	:= iStep + 10;		
	160	:	//pierwszy krok 
		AssertTrue (Condition := GVL_TestSaMContoller.fbMySaMController.IsChangeStateBusy (), 		Message := 'S160 - T01 - Bledny stan busy');
		AssertFalse (Condition := GVL_TestSaMContoller.fbMySaMController.IsChangeStateDone (), 		Message := 'S160 - T02 - Bledny stan done');
		AssertFalse (Condition := GVL_TestSaMContoller.fbMySaMController.IsChangeStateStatus (), 	Message := 'S160 - T03 - Bledny stan status');
		iStep	:= iStep + 10;
	170	://krok zmiany stanu
		AssertTrue (Condition := GVL_TestSaMContoller.fbMySaMController.IsChangeStateBusy (), 		Message := 'S170 - T01 - Bledny stan busy');
		AssertFalse (Condition := GVL_TestSaMContoller.fbMySaMController.IsChangeStateDone (),		Message := 'S170 - T02 - Bledny stan done');
		AssertFalse (Condition := GVL_TestSaMContoller.fbMySaMController.IsChangeStateStatus (), 	Message := 'S170 - T03 - Bledny stan status');
		iStep	:= iStep + 10;
	180	:	//ostani krok 
		AssertFalse (Condition := GVL_TestSaMContoller.fbMySaMController.IsChangeStateBusy (), 		Message := 'S180 - T01 - Bledny stan busy');
		AssertTrue (Condition := GVL_TestSaMContoller.fbMySaMController.IsChangeStateDone (), 		Message := 'S180 - T02 - Bledny stan done');
		AssertTrue (Condition := GVL_TestSaMContoller.fbMySaMController.IsChangeStateStatus (), 	Message := 'S180 - T03 - Bledny stan status');
		eActualState				:= GVL_TestSaMContoller.fbMySaMController.GetState ();
		AssertEquals (Expected := eNewState, Actual := eActualState, 						Message := 'S180 - T04 - Bledny stan');
		iStep	:= iStep + 10;
	190	:	//przjescie do aborting
(*	*)	eNewState			:= E_BaseMachineState.Aborting;
		GVL_TestSaMContoller.fbMySaMController.Execute (iNumberOfCommand := E_SaMCommandChangeState.Abort, eChangeCategory := E_SaMChangeCategory.eState);
		iStep	:= iStep + 10;
	200	:	//pierwszy krok 
		AssertTrue (Condition := GVL_TestSaMContoller.fbMySaMController.IsChangeStateBusy (), 		Message := 'S200 - T01 - Bledny stan busy');
		AssertFalse (Condition := GVL_TestSaMContoller.fbMySaMController.IsChangeStateDone (), 		Message := 'S200 - T02 - Bledny stan done');
		AssertFalse (Condition := GVL_TestSaMContoller.fbMySaMController.IsChangeStateStatus (), 	Message := 'S200 - T03 - Bledny stan status');
		iStep	:= iStep + 10;
	210	://krok zmiany stanu
		AssertTrue (Condition := GVL_TestSaMContoller.fbMySaMController.IsChangeStateBusy (), 		Message := 'S210 - T01 - Bledny stan busy');
		AssertFalse (Condition := GVL_TestSaMContoller.fbMySaMController.IsChangeStateDone (),		Message := 'S210 - T02 - Bledny stan done');
		AssertFalse (Condition := GVL_TestSaMContoller.fbMySaMController.IsChangeStateStatus (), 	Message := 'S210 - T03 - Bledny stan status');
		iStep	:= iStep + 10;
	220	:	//ostani krok 
		AssertFalse (Condition := GVL_TestSaMContoller.fbMySaMController.IsChangeStateBusy (), 		Message := 'S220 - T01 - Bledny stan busy');
		AssertTrue (Condition := GVL_TestSaMContoller.fbMySaMController.IsChangeStateDone (), 		Message := 'S220 - T02 - Bledny stan done');
		AssertTrue (Condition := GVL_TestSaMContoller.fbMySaMController.IsChangeStateStatus (), 	Message := 'S220 - T03 - Bledny stan status');
		eActualState				:= GVL_TestSaMContoller.fbMySaMController.GetState ();
		AssertEquals (Expected := eNewState, Actual := eActualState, 						Message := 'S220 - T04 - Bledny stan');
		iStep	:= iStep + 10;
	230	:
		iStep	:= iStep + 10;
	240	:	
(*	*)	eNewState			:= E_BaseMachineState.Aborted;
		GVL_TestSaMContoller.fbMySaMController.ChangeStateTo (eNewState := eNewState);
		iStep	:= iStep + 10;		
	250	:	//pierwszy krok 
		AssertTrue (Condition := GVL_TestSaMContoller.fbMySaMController.IsChangeStateBusy (), 		Message := 'S250 - T01 - Bledny stan busy');
		AssertFalse (Condition := GVL_TestSaMContoller.fbMySaMController.IsChangeStateDone (), 		Message := 'S250 - T02 - Bledny stan done');
		AssertFalse (Condition := GVL_TestSaMContoller.fbMySaMController.IsChangeStateStatus (), 	Message := 'S250 - T03 - Bledny stan status');
		iStep	:= iStep + 10;
	260	://krok zmiany stanu
		AssertTrue (Condition := GVL_TestSaMContoller.fbMySaMController.IsChangeStateBusy (), 		Message := 'S260 - T01 - Bledny stan busy');
		AssertFalse (Condition := GVL_TestSaMContoller.fbMySaMController.IsChangeStateDone (),		Message := 'S260 - T02 - Bledny stan done');
		AssertFalse (Condition := GVL_TestSaMContoller.fbMySaMController.IsChangeStateStatus (), 	Message := 'S260 - T03 - Bledny stan status');
		iStep	:= iStep + 10;
	270	:	//ostani krok 
		AssertFalse (Condition := GVL_TestSaMContoller.fbMySaMController.IsChangeStateBusy (), 		Message := 'S270 - T01 - Bledny stan busy');
		AssertTrue (Condition := GVL_TestSaMContoller.fbMySaMController.IsChangeStateDone (), 		Message := 'S270 - T02 - Bledny stan done');
		AssertTrue (Condition := GVL_TestSaMContoller.fbMySaMController.IsChangeStateStatus (), 	Message := 'S270 - T03 - Bledny stan status');
		eActualState				:= GVL_TestSaMContoller.fbMySaMController.GetState ();
		AssertEquals (Expected := eNewState, Actual := eActualState, 						Message := 'S270 - T04 - Bledny stan');
		iStep	:= iStep + 10;
	280	:
		GVL_TestSaMContoller.fbMySaMController.SetStateEnabledInMode (iMode := E_BaseMachineMode.Production, iState := E_BaseMachineState.Clearing, bValue := FALSE);
		iStep	:= iStep + 10;
	290	:
(*	*)	eNewState			:= E_BaseMachineState.Clearing;
		GVL_TestSaMContoller.fbMySaMController.Execute (iNumberOfCommand := E_SaMCommandChangeState.Clear, eChangeCategory := E_SaMChangeCategory.eState);
		iStep	:= iStep + 10;
	300	:	//pierwszy krok 
		AssertFalse (Condition := GVL_TestSaMContoller.fbMySaMController.IsChangeStateBusy (), 		Message := 'S300 - T01 - Bledny stan busy');
		AssertTrue (Condition := GVL_TestSaMContoller.fbMySaMController.IsChangeStateDone (), 		Message := 'S300 - T02 - Bledny stan done');
		AssertTrue (Condition := GVL_TestSaMContoller.fbMySaMController.IsChangeStateStatus (), 	Message := 'S300 - T03 - Bledny stan status');
		iStep	:= iStep + 10;
	310	:
		GVL_TestSaMContoller.fbMySaMController.SetStateEnabledInMode (iMode := E_BaseMachineMode.Production, iState := E_BaseMachineState.Clearing, bValue := TRUE);
		iStep	:= iStep + 10;
	320	:
(*	*)	eNewState			:= E_BaseMachineState.Clearing;
		GVL_TestSaMContoller.fbMySaMController.Execute (iNumberOfCommand := E_SaMCommandChangeState.Clear, eChangeCategory := E_SaMChangeCategory.eState);
		iStep	:= iStep + 10;
	330	:	//pierwszy krok 
		AssertTrue (Condition := GVL_TestSaMContoller.fbMySaMController.IsChangeStateBusy (), 		Message := 'S330 - T01 - Bledny stan busy');
		AssertFalse (Condition := GVL_TestSaMContoller.fbMySaMController.IsChangeStateDone (), 		Message := 'S330 - T02 - Bledny stan done');
		AssertFalse (Condition := GVL_TestSaMContoller.fbMySaMController.IsChangeStateStatus (), 	Message := 'S330 - T03 - Bledny stan status');
		iStep	:= iStep + 10;
	340	://krok zmiany stanu
		AssertTrue (Condition := GVL_TestSaMContoller.fbMySaMController.IsChangeStateBusy (), 		Message := 'S340 - T01 - Bledny stan busy');
		AssertFalse (Condition := GVL_TestSaMContoller.fbMySaMController.IsChangeStateDone (),		Message := 'S340 - T02 - Bledny stan done');
		AssertFalse (Condition := GVL_TestSaMContoller.fbMySaMController.IsChangeStateStatus (), 	Message := 'S340 - T03 - Bledny stan status');
		iStep	:= iStep + 10;
	350	:	//ostani krok 
		AssertFalse (Condition := GVL_TestSaMContoller.fbMySaMController.IsChangeStateBusy (), 		Message := 'S350 - T01 - Bledny stan busy');
		AssertTrue (Condition := GVL_TestSaMContoller.fbMySaMController.IsChangeStateDone (), 		Message := 'S350 - T02 - Bledny stan done');
		AssertTrue (Condition := GVL_TestSaMContoller.fbMySaMController.IsChangeStateStatus (), 	Message := 'S350 - T03 - Bledny stan status');
		eActualState				:= GVL_TestSaMContoller.fbMySaMController.GetState ();
		AssertEquals (Expected := eNewState, Actual := eActualState, 						Message := 'S350 - T04 - Bledny stan');
		iStep	:= iStep + 10;
	360	:
		TcUnit.TEST_FINISHED ();
	END_CASE
END_IF
END_METHOD

END_FUNCTION_BLOCK
